(* IEC 61131-3 sources: CodesysTest/alpha/export/Pro18_1174_04.dev/Plc Logic/Application/Motors/Applied Motion/FB_AppliedMotionBagDeliveryMotor_1.pou, 3 files *)

(* ---- FB_AppliedMotionBagDeliveryMotor_1.pou.st ---- *)
(*#-#-#-#-#-#-#-#-#-#---Declaration---#-#-#-#-#-#-#-#-#-#-#-#-#*)

FUNCTION_BLOCK FB_AppliedMotionBagDeliveryMotor_1 EXTENDS FB_AppliedMotionStepServoEIPBase
VAR_INPUT
END_VAR
VAR_OUTPUT
END_VAR
VAR
	_moveDistance : BOOL;
	_moveDistanceONS : R_TRIG;
	_moveFinal : BOOL;
	_moveFinalONS : R_TRIG;
	_moveDone : BOOL;
	waitForMove : TON := (PT := T#30MS);
	manualFinalMovePB : BOOL;
	movedFinal : BOOL;
	moveDistanceState : BAG_DELIVERY_MOVE_STATES;
	moveDistanceFinalState : BAG_DELIVERY_MOVE_STATES;
END_VAR
(*#-#-#-#-#-#-#-#-#-#---Implementation---#-#-#-#-#-#-#-#-#-#-#-#-#*)

(* ---- Execute.m.st ---- *)
(*#-#-#-#-#-#-#-#-#-#---Declaration---#-#-#-#-#-#-#-#-#-#-#-#-#*)

METHOD Execute
VAR_INPUT
END_VAR
(*#-#-#-#-#-#-#-#-#-#---Implementation---#-#-#-#-#-#-#-#-#-#-#-#-#*)

SUPER^.Execute();
waitForMove();
_moveDistanceONS(CLK := _moveDistance);
_moveFinalONS(CLK := _moveFinal);

CASE moveDistanceState OF
	BAG_DELIVERY_MOVE_STATES.Idle :
															IF _moveDistance THEN
																moveDistanceState := BAG_DELIVERY_MOVE_STATES.SetToPointToPointMode;
															END_IF

	BAG_DELIVERY_MOVE_STATES.SetToPointToPointMode :					sclCommand := 16#534F; //Output off
															parameter1 := 16#48B2;
															commands.SendHostCommand := TRUE;
															IF commandSuccessful THEN
																commandSuccessful := FALSE;
																moveDistanceState := BAG_DELIVERY_MOVE_STATES.WaitAfterSettingOutputOff;
															END_IF

	BAG_DELIVERY_MOVE_STATES.WaitAfterSettingOutputOff :
															IF commandSuccessful THEN
																moveDistanceState := BAG_DELIVERY_MOVE_STATES.MoveMotor;
															END_IF

	BAG_DELIVERY_MOVE_STATES.MoveMotor: 					commandSuccessful := FALSE;
															sclCommand := 16#0;
															parameter1 := 16#0;
															commands.FeedToLength := TRUE;
															_moveDistance := FALSE;
															moveDistanceState := BAG_DELIVERY_MOVE_STATES.WaitAfterMovingMotor;

	BAG_DELIVERY_MOVE_STATES.WaitAfterMovingMotor: 		IF commandSuccessful THEN
																_moveDone := TRUE;
																moveDistanceState := BAG_DELIVERY_MOVE_STATES.Idle;
															END_IF
END_CASE

CASE moveDistanceFinalState OF
	BAG_DELIVERY_MOVE_STATES.Idle :						IF _moveFinal THEN
																moveDistanceFinalState := BAG_DELIVERY_MOVE_STATES.SetToPointToPointMode;
															END_IF

	BAG_DELIVERY_MOVE_STATES.SetToPointToPointMode :					sclCommand := 16#534F; //Output off
															parameter1 := 16#48B2;
															commands.SendHostCommand := TRUE;
															IF commandSuccessful THEN
																commandSuccessful := FALSE;
																moveDistanceFinalState := BAG_DELIVERY_MOVE_STATES.WaitAfterSettingOutputOff;
															END_IF

	BAG_DELIVERY_MOVE_STATES.WaitAfterSettingOutputOff :
															IF commandSuccessful THEN
																moveDistanceFinalState := BAG_DELIVERY_MOVE_STATES.MoveMotor;
															END_IF

	BAG_DELIVERY_MOVE_STATES.MoveMotor: 					sclCommand := 16#0;
															parameter1 := 16#0;
															commandSuccessful := FALSE;
															commands.FeedToLength := TRUE;
															moveDistanceFinalState := BAG_DELIVERY_MOVE_STATES.WaitAfterMovingMotor;

	BAG_DELIVERY_MOVE_STATES.WaitAfterMovingMotor: 		IF commandSuccessful AND InPosition THEN
																moveDistanceFinalState := BAG_DELIVERY_MOVE_STATES.SetToTorqueMode;
															END_IF

	BAG_DELIVERY_MOVE_STATES.SetToTorqueMode :					sclCommand := 16#534F; // Output on
															parameter1 := 16#4CB2;

															commandSuccessful := FALSE;
															commands.SendHostCommand := TRUE;
															_moveFinal := FALSE;
															moveDistanceFinalState := BAG_DELIVERY_MOVE_STATES.WaitAfterSettingOutputOn;

	BAG_DELIVERY_MOVE_STATES.WaitAfterSettingOutputOn :
															IF commandSuccessful THEN
																_moveDone := TRUE;
																moveDistanceFinalState := BAG_DELIVERY_MOVE_STATES.Idle;
															END_IF

END_CASE
(*
IF _moveFinal THEN
	IF NOT movedFinal AND commandSuccessful THEN
		commandSuccessful := FALSE;
		commands.FeedToLength := TRUE;
		waitForMove.IN := TRUE;
		movedFinal := TRUE;
	END_IF

	IF commandSuccessful AND waitForMove.Q AND InPosition THEN
		sclCommand := 16#534F;
		parameter1 := 16#4CB2;
		commands.SendHostCommand := TRUE;
		_moveFinal := FALSE;
		waitForMove.IN := FALSE;
		movedFinal := FALSE;
	END_IF
END_IF
*)
IF manualFinalMovePB THEN
    MoveDistanceFinal(distance := distanceSetpointInches, acceleration := pointToPointAccelSetpoint, deceleration := pointToPointDecelSetpoint, velocity := velocitySetpoint);
    manualFinalMovePB := FALSE;
END_IF

(* ---- MoveDistanceFinal.m.st ---- *)
(*#-#-#-#-#-#-#-#-#-#---Declaration---#-#-#-#-#-#-#-#-#-#-#-#-#*)

METHOD MoveDistanceFinal
VAR_INPUT
    distance : REAL;        //Distance to move in inches
    acceleration : INT;        //Acceleration in RPM/sec
    deceleration : INT;        //Deceleration in RPM/sec
    velocity : INT;            //Velocity in .25RPM
END_VAR
(*#-#-#-#-#-#-#-#-#-#---Implementation---#-#-#-#-#-#-#-#-#-#-#-#-#*)

commandSuccessful := FALSE;
_moveDone := FALSE;
moveDistanceFinalState := BAG_DELIVERY_MOVE_STATES.Idle;
distanceToMoveInSteps := REAL_TO_DINT((distance) * stepsPerInchSetpoint);
IF reversePolarity THEN
    distanceToMoveInSteps := distanceToMoveInSteps * -1;
END_IF

pointToPointAccelSetpoint := acceleration;
pointToPointDecelSetpoint := deceleration;
velocitySetpoint := velocity;

currentLimit := defaultCurrentSetpoint;
_moveFinal := TRUE;
//SUPER^.ExecuteStoredProgram(2);
